FUNCTION IArgToIRoom : Result
VAR_INPUT
	iSource	: I_Arg;
END_VAR
VAR_OUTPUT
	iDest	: I_Room;
END_VAR

IF iSource = 0 THEN
	IArgToIRoom := Err.Itf0;
	RETURN;
END_IF

IF __QUERYINTERFACE(iSource, iDest) THEN
	IArgToIRoom := Ok;
ELSE
	iDest := 0;
	IArgToIRoom := Err.NoMatch;
END_IF

END_FUNCTION

(* stored: Version 1.1.0.1
   POU IArgToIRoom: Id {d00b227c-37ec-41f5-802c-208b27ba6260}, SpecialFunc None *)
